{attribute 'no_explicit_call' := 'LightOnCommand is a CLASS and must be accessed using methods or properties'}
FUNCTION_BLOCK OpenCommand IMPLEMENTS I_Command
VAR
	_openCommand					: I_OpenCommand;
END_VAR


// The body of a class must not be used for code.  
// Cyclic code should be called from a method if needed.

METHOD Execute
_openCommand.Open();
END_METHOD

METHOD FB_init : BOOL
VAR_INPUT
	bInitRetains : BOOL; // if TRUE, the retain variables are initialized (warm start / cold start)
	bInCopyCode : BOOL;  // if TRUE, the instance afterwards gets moved into the copy code (online change)
	OpenCommand			: I_OpenCommand;
END_VAR
_openCommand  := OpenCommand;
END_METHOD

END_FUNCTION_BLOCK

(* stored: Version 1.1.0.1, ProductVersion 3.1.4024.11
   POU OpenCommand: Id {06e37c97-b385-4b71-88be-a813cdd6d696}, SpecialFunc None
   Method Execute: Id {2b5750eb-b1f8-41ec-bcbe-111a53a2e971}
   Method FB_init: Id {6344836e-a82a-4d73-ad80-1380aeded92f} *)
